FUNCTION_BLOCK FB_PowerNC IMPLEMENTS I_Power
VAR
    {attribute 'no_copy'}
    AxisRef : REFERENCE TO AXIS_REF;
    fbMcPower : MC_Power;

END_VAR

IF NOT __ISVALIDREF(AxisRef) THEN
    RETURN;
END_IF

AxisRef.ReadStatus();

fbMcPower(
    Axis := AxisRef,
);

PROPERTY Busy : BOOL
GET
Busy := THIS^.fbMcPower.Busy;
END_GET
END_PROPERTY

METHOD PUBLIC CallAfterInit
VAR_INPUT
    AxisRef : REFERENCE TO AXIS_REF;
END_VAR
THIS^.AxisRef REF= AxisRef;
END_METHOD

{warning 'Add method implementation '}
METHOD DisablePower
(*Use to remove power in DURING_MOTION driving mode *)
THIS^.fbMcPower(
    Axis := THIS^.AxisRef,
    Enable := FALSE
);
END_METHOD

PROPERTY Done : BOOL
GET
END_GET
END_PROPERTY

PROPERTY Error : BOOL
GET
Error := THIS^.fbMcPower.Error;
END_GET
END_PROPERTY

PROPERTY ErrorID : UDINT
GET
ErrorID := THIS^.fbMcPower.ErrorID;
END_GET
END_PROPERTY

//FB_Init is always available implicitly and it is used primarily for initialization.
//The return value is not evaluated. For a specific influence, you can also declare the
//methods explicitly and provide additional code there with the standard initialization
//code. You can evaluate the return value.
METHOD FB_Init: BOOL
VAR_INPUT
    bInitRetains: BOOL; // TRUE: the retain variables are initialized (reset warm / reset cold)
    bInCopyCode: BOOL;  // TRUE: the instance will be copied to the copy code afterward (online change)
    AxisRef : REFERENCE TO AXIS_REF;
END_VAR
THIS^.AxisRef REF= AxisRef;
END_METHOD

PROPERTY Message : T_MAXSTRING
GET
END_GET
END_PROPERTY

PROPERTY Override : LREAL
GET
Override := THIS^.fbMcPower.Override;
END_GET
END_PROPERTY

(*When the enable flags are updated externally this must be called cyclicly*)
METHOD Power
VAR_INPUT
    Enable	: BOOL;
    Enable_Positive	: BOOL;
    Enable_Negative	: BOOL;
    Override	: LREAL := 100.0;
    BufferMode	: MC_BufferMode := MC_BufferMode.MC_Aborting;
END_VAR
(*The calling block must provide homing directional Power enables override *)
THIS^.fbMcPower(
    Axis := THIS^.AxisRef,
    Enable := Enable,
    Enable_Positive := Enable_Positive,
    Enable_Negative := Enable_Negative,
    BufferMode := BufferMode,
    Override :=Override
);
END_METHOD

PROPERTY PowerIsEnabled : BOOL
GET
PowerIsEnabled :=THIS^.fbMcPower.Status;
END_GET
END_PROPERTY

END_FUNCTION_BLOCK

(* stored: Version 1.1.0.1
   POU FB_PowerNC: Id {82bac45d-f3fb-4090-96f5-9cec57f017c8}, SpecialFunc None
   Property Busy: Id {1d88cc85-9bbc-4836-b583-4a9d93ccadc7}
   Get Get: Id {e8b60715-a1d9-4e57-9f76-50ea68243628}
   Method CallAfterInit: Id {b807f150-fc9f-4aa5-9d8d-b294c818c5aa}
   Method DisablePower: Id {577374a6-9c8d-40f0-8c0b-b6bac87de3d0}
   Property Done: Id {47775ab2-32ed-415e-8f00-7dc8c50e6589}
   Get Get: Id {8a26bdf6-610d-44e7-af87-ff96e882b31e}
   Property Error: Id {5900c701-bb24-4682-9d2c-47b8d2773b46}
   Get Get: Id {50fb1906-033c-485b-9e5d-f1230f94dfc8}
   Property ErrorID: Id {1fe914ad-7f24-41a0-bde2-d4d693aeb73f}
   Get Get: Id {8f8eef06-c2be-4844-866a-ef0542739cd8}
   Method FB_Init: Id {cf7caa46-f1e4-49f9-addf-eba93ec02164}
   Property Message: Id {8449188f-1930-49b3-8fe2-2e40bd14ae5f}
   Get Get: Id {1b9ef192-6b77-407c-a88f-8d85eb8cdc1a}
   Property Override: Id {a7a1e83f-16ea-4038-8048-9acd1171492b}
   Get Get: Id {c098132b-e311-41da-b640-f143b09d83d2}
   Method Power: Id {b859403c-f315-4c59-bb46-554245f47326}
   Property PowerIsEnabled: Id {7e136934-4440-48f5-a211-011704d8f4f5}
   Get Get: Id {fffb35ff-b9f5-44f8-bd6c-842b697893c4} *)
